TYPE ST_CommunicationConfig :
STRUCT

    sIpAddress : STRING(15) := '192.168.0.10';
    nPort : UINT := 7171;
	sUsername: STRING(128):= '';
    sPassword : STRING(128) := '';
    tTimeout : TIME := T#5S;
    bAutoReconnect : BOOL := TRUE;
END_STRUCT
END_TYPE

(* stored: Version 1.1.0.1, ProductVersion 3.1.4026.18
   DUT ST_CommunicationConfig: Id {30496dbe-ef77-43fa-a92a-f084f7770640} *)
